// TIA Portal V18 export
FUNCTION "DOadv" : Void   // FC10009, LAD
{ S7_Optimized_Access := 'TRUE' }
VERSION : 0.1
// stored: AutoNumber false, IsIECCheckEnabled false, SetENOAutomatically false, UDAEnableTagReadback false
   VAR_INPUT
      xInput : Bool;
      xInversion : Bool;   // 0-direct / 1-reverse
      cMOA : Byte;
   END_VAR
   VAR_OUTPUT
      xOutput : Bool;
   END_VAR
   VAR_IN_OUT
      xMemoryOut : Bool;
      xMemoryIn : Bool;
      cMemory : Byte;
      iCounterIn : Int;
      iCounterOut : Int;
   END_VAR
   VAR_TEMP
      InOut_1 : Bool;
   END_VAR
BEGIN

REGION Network 1 (SCL)
   CASE #cMOA OF
       0: // OFF
           #xOutput := FALSE;

       1: // MANUAL
           #xOutput := TRUE;

       2: // AUTO
           #xOutput :=#xInput;

   ELSE
       #xOutput := FALSE;
   END_CASE;
END_REGION

REGION Network 2 (SCL)
   IF #xInversion THEN
       #xOutput := NOT #xOutput;
   END_IF;
END_REGION

REGION Network 3 (SCL)
   IF (#xMemoryIn XOR #xInput) THEN
       IF #iCounterIn > 30000 THEN
           #iCounterIn := 5;
       ELSE
           #iCounterIn := #iCounterIn + 1;
       END_IF;
   END_IF;
   #xMemoryIn := #xInput;
END_REGION

REGION Network 4 (SCL)
   IF (#xMemoryOut XOR #xOutput) THEN
       IF #iCounterOut > 30000 THEN
           #iCounterOut := 5;
       ELSE
           #iCounterOut := #iCounterOut + 1;
       END_IF;
   END_IF;
   #xMemoryOut := #xOutput;
END_REGION
END_FUNCTION
